(* Schneider Machine Expert - Basic project taffic_control_project, file version 1.8.0.0 *)
(* ProjectInformations: Name=New project *)

HARDWARE
  Cpu 0: TM221CE16R
  EthernetConfiguration: NetworkName=M221, IpAllocationMode=FixedAddress, IpAddress=0.0.0.0, SubnetMask=0.0.0.0
  SerialLineConfiguration: Baud=Baud19200, Parity=ParityEven, DataBits=DataBits8, StopBits=StopBits1, PhysicalMedium=PhysicalMediumRs485, TransmissionMode=TransmissionModeModbusRtu, SlaveId=1, Addressing=SlaveAddressing
  MastTask: UsePeriodScanMode=false, PeriodScan=100
  FastTask: Period=255
  CpuBehavior: StartingMode=StartAsPreviousState, AutoSaveRamOnEeprom=true, WatchdogPeriod=250

SYMBOLS  (address, symbol, comment, settings)
  %TM0        [Preset=1, Base=OneSecond, IsRetentive=true]
  %TM1        [Preset=1, Base=OneSecond, IsRetentive=true]
  %TM2        [Preset=5, Base=OneSecond, IsRetentive=true]
  %TM3        [Preset=3, Base=OneSecond, IsRetentive=true]
  %TM4        [Preset=3, Base=OneSecond, IsRetentive=true]
  %TM5        [Preset=3, Base=OneSecond, IsRetentive=true]
  %TM6        [Preset=3, Base=OneSecond, IsRetentive=true]

POU state
  (* SectionNumber=1 *)

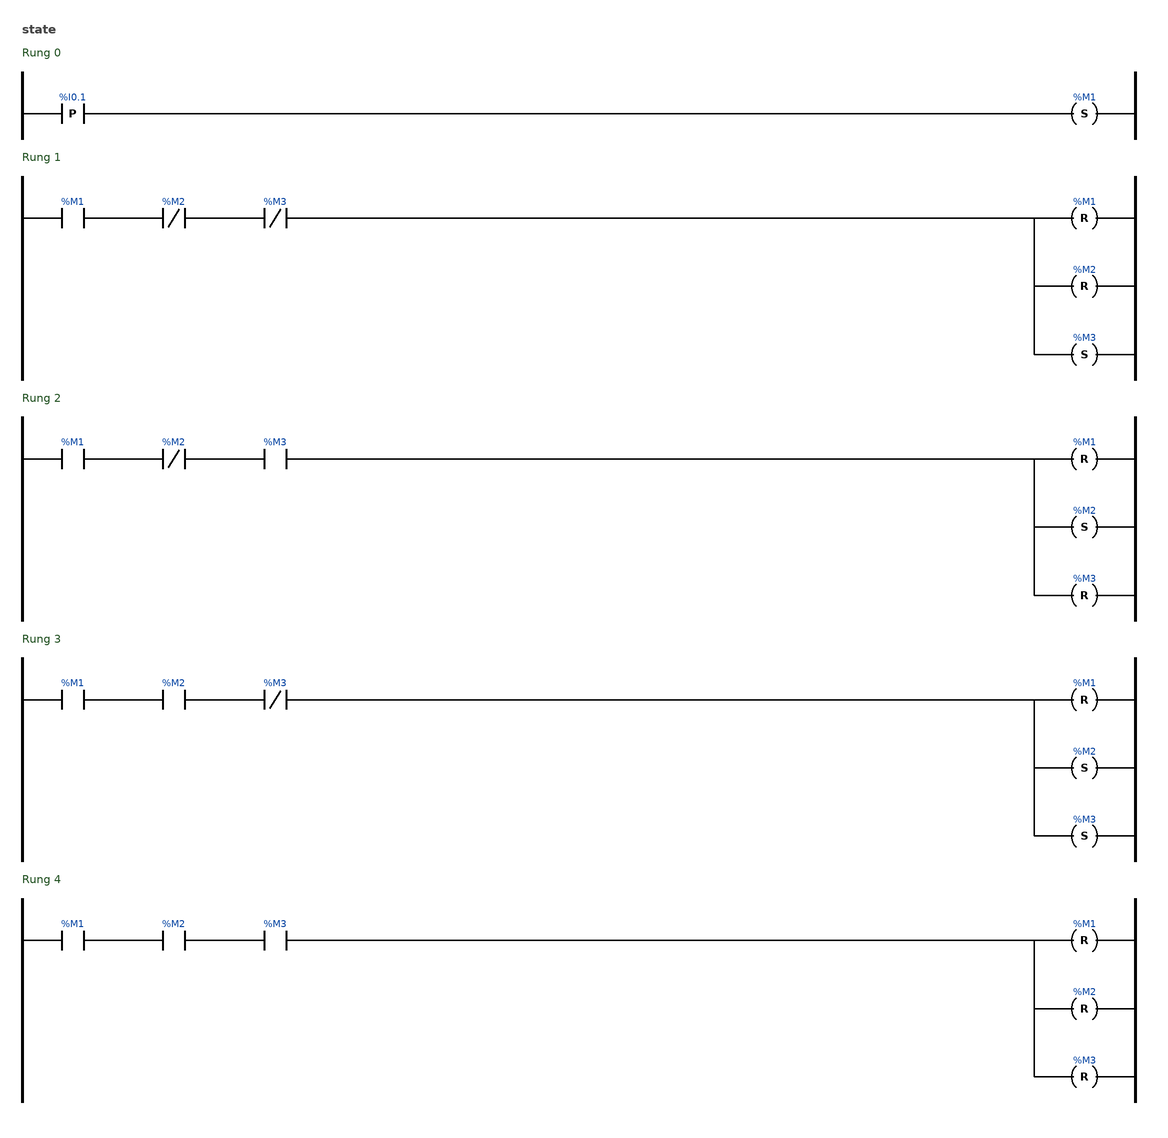

// Rung 0
  LDR %I0.1
  S %M1
  // as ST:
  //   IF RISING(%I0.1) THEN %M1 := TRUE; END_IF;

// Rung 1
  LD %M1
  ANDN %M2
  ANDN %M3
  R %M1
  R %M2
  S %M3
  // as ST:
  //   _t1 := %M1 AND NOT %M2 AND NOT %M3;
  //   IF _t1 THEN %M1 := FALSE; END_IF;
  //   IF _t1 THEN %M2 := FALSE; END_IF;
  //   IF _t1 THEN %M3 := TRUE; END_IF;

// Rung 2
  LD %M1
  ANDN %M2
  AND %M3
  R %M1
  S %M2
  R %M3
  // as ST:
  //   _t1 := %M1 AND NOT %M2 AND %M3;
  //   IF _t1 THEN %M1 := FALSE; END_IF;
  //   IF _t1 THEN %M2 := TRUE; END_IF;
  //   IF _t1 THEN %M3 := FALSE; END_IF;

// Rung 3
  LD %M1
  AND %M2
  ANDN %M3
  R %M1
  S %M2
  S %M3
  // as ST:
  //   _t1 := %M1 AND %M2 AND NOT %M3;
  //   IF _t1 THEN %M1 := FALSE; END_IF;
  //   IF _t1 THEN %M2 := TRUE; END_IF;
  //   IF _t1 THEN %M3 := TRUE; END_IF;

// Rung 4
  LD %M1
  AND %M2
  AND %M3
  R %M1
  R %M2
  R %M3
  // as ST:
  //   _t1 := %M1 AND %M2 AND %M3;
  //   IF _t1 THEN %M1 := FALSE; END_IF;
  //   IF _t1 THEN %M2 := FALSE; END_IF;
  //   IF _t1 THEN %M3 := FALSE; END_IF;

POU yello blink
  (* SectionNumber=2 *)

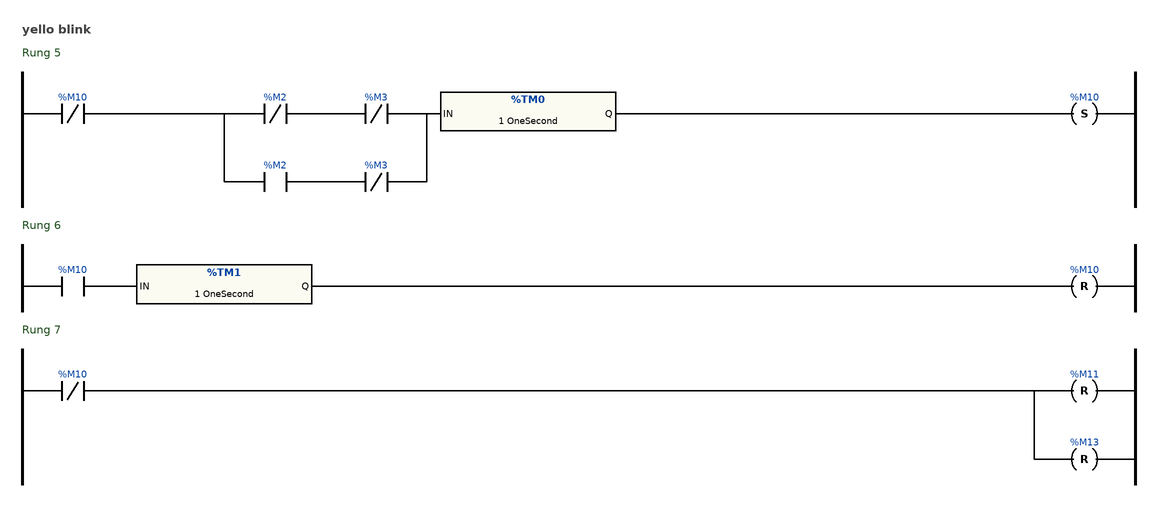

// Rung 5
  BLK %TM0
  LDN %M10
  AND(N %M2
  ANDN %M3
  OR( %M2
  ANDN %M3
  )
  )
  IN
  OUT_BLK
  LD Q
  S %M10
  END_BLK
  // as ST:
  //   %TM0(IN := NOT %M10 AND (NOT %M2 AND NOT %M3 OR %M2 AND NOT %M3));
  //   IF %TM0.Q THEN %M10 := TRUE; END_IF;

// Rung 6
  BLK %TM1
  LD %M10
  IN
  OUT_BLK
  LD Q
  R %M10
  END_BLK
  // as ST:
  //   %TM1(IN := %M10);
  //   IF %TM1.Q THEN %M10 := FALSE; END_IF;

// Rung 7
  LDN %M10
  R %M11
  R %M13
  // as ST:
  //   IF NOT %M10 THEN %M11 := FALSE; END_IF;
  //   IF NOT %M10 THEN %M13 := FALSE; END_IF;

POU Manual
  (* SectionNumber=3 *)

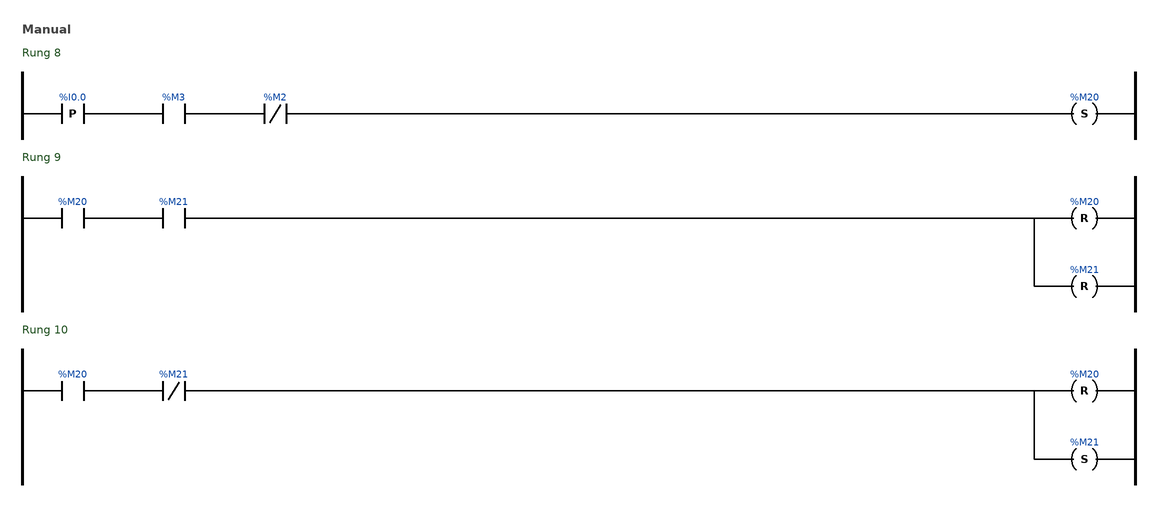

// Rung 8
  LDR %I0.0
  AND %M3
  ANDN %M2
  S %M20
  // as ST:
  //   IF RISING(%I0.0) AND %M3 AND NOT %M2 THEN %M20 := TRUE; END_IF;

// Rung 9
  LD %M20
  AND %M21
  R %M20
  R %M21
  // as ST:
  //   _t1 := %M20 AND %M21;
  //   IF _t1 THEN %M20 := FALSE; END_IF;
  //   IF _t1 THEN %M21 := FALSE; END_IF;

// Rung 10
  LD %M20
  ANDN %M21
  R %M20
  S %M21
  // as ST:
  //   _t1 := %M20 AND NOT %M21;
  //   IF _t1 THEN %M20 := FALSE; END_IF;
  //   IF _t1 THEN %M21 := TRUE; END_IF;

POU Manual_LED
  (* SectionNumber=4 *)

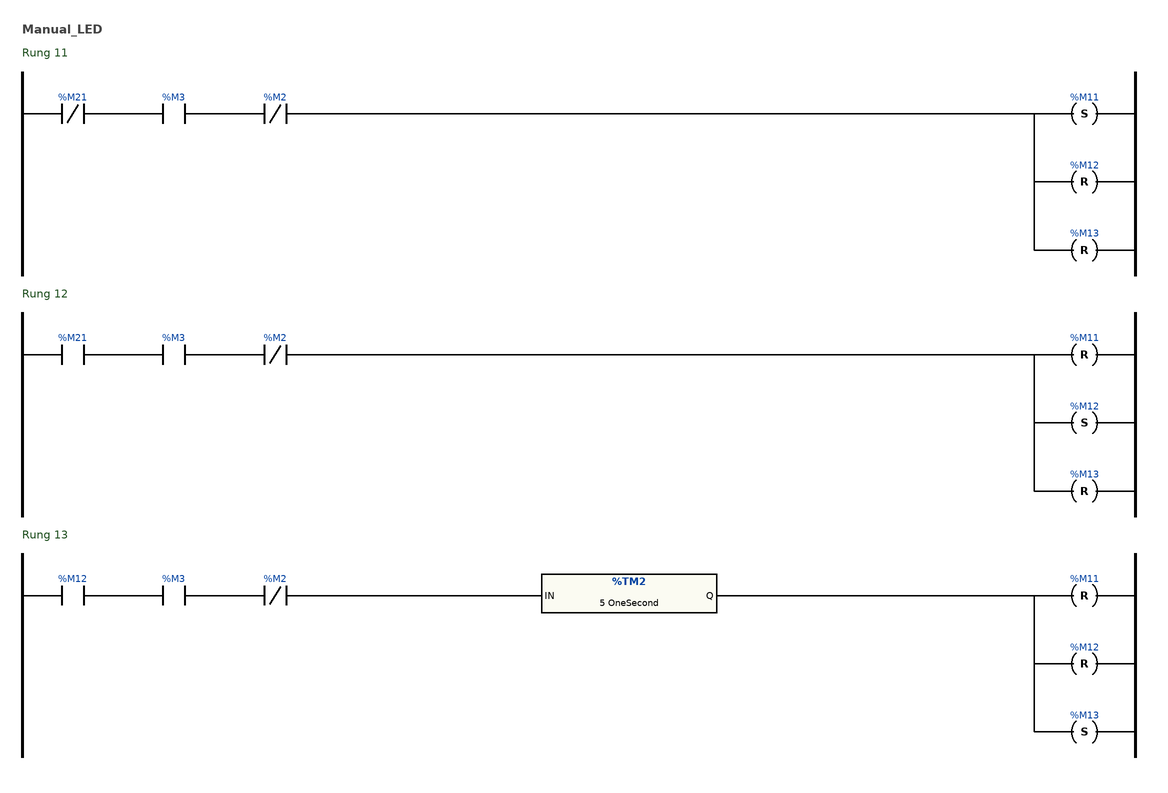

// Rung 11
  LDN %M21
  AND %M3
  ANDN %M2
  S %M11
  R %M12
  R %M13
  // as ST:
  //   IF NOT %M21 AND %M3 AND NOT %M2 THEN %M11 := TRUE; END_IF;
  //   IF NOT %M21 AND %M3 AND NOT %M2 THEN %M12 := FALSE; END_IF;
  //   IF NOT %M21 AND %M3 AND NOT %M2 THEN %M13 := FALSE; END_IF;

// Rung 12
  LD %M21
  AND %M3
  ANDN %M2
  R %M11
  S %M12
  R %M13
  // as ST:
  //   IF %M21 AND %M3 AND NOT %M2 THEN %M11 := FALSE; END_IF;
  //   IF %M21 AND %M3 AND NOT %M2 THEN %M12 := TRUE; END_IF;
  //   IF %M21 AND %M3 AND NOT %M2 THEN %M13 := FALSE; END_IF;

// Rung 13
  BLK %TM2
  LD %M12
  AND %M3
  ANDN %M2
  IN
  OUT_BLK
  LD Q
  R %M11
  R %M12
  S %M13
  END_BLK
  // as ST:
  //   %TM2(IN := %M12 AND %M3 AND NOT %M2);
  //   IF %TM2.Q THEN %M11 := FALSE; END_IF;
  //   IF %TM2.Q THEN %M12 := FALSE; END_IF;
  //   IF %TM2.Q THEN %M13 := TRUE; END_IF;

POU LED_Control
  (* SectionNumber=5 *)

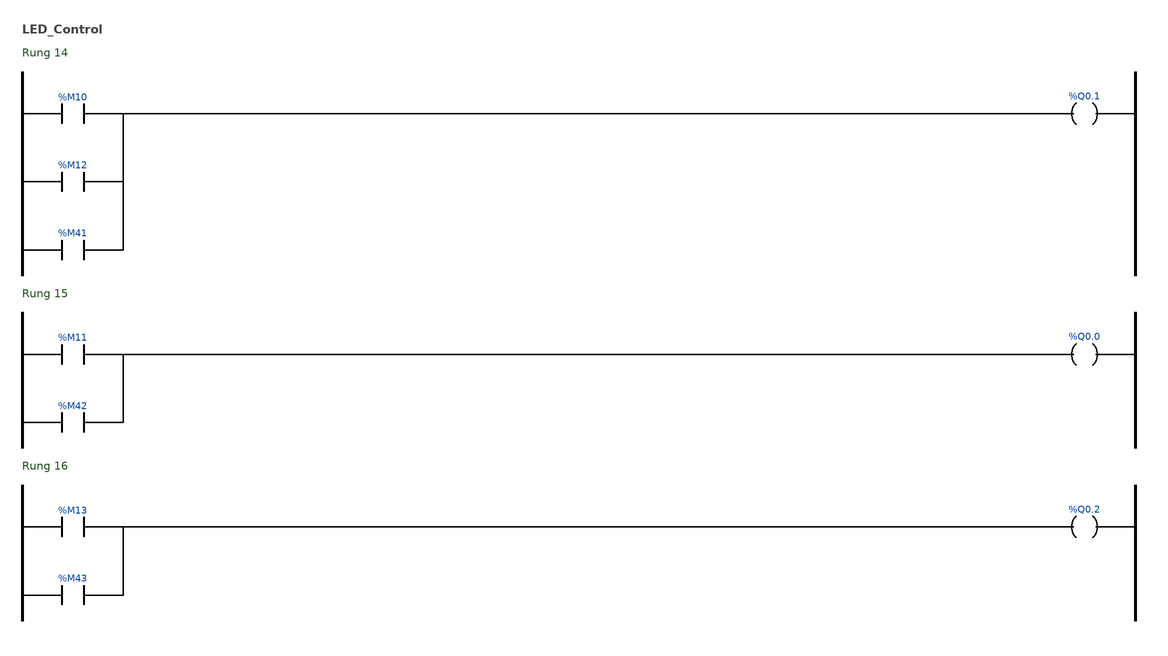

// Rung 14
  LD %M10
  OR %M12
  OR %M41
  ST %Q0.1
  // as ST:
  //   %Q0.1 := %M10 OR %M12 OR %M41;

// Rung 15
  LD %M11
  OR %M42
  ST %Q0.0
  // as ST:
  //   %Q0.0 := %M11 OR %M42;

// Rung 16
  LD %M13
  OR %M43
  ST %Q0.2
  // as ST:
  //   %Q0.2 := %M13 OR %M43;

POU Auto_Control
  (* SectionNumber=6 *)

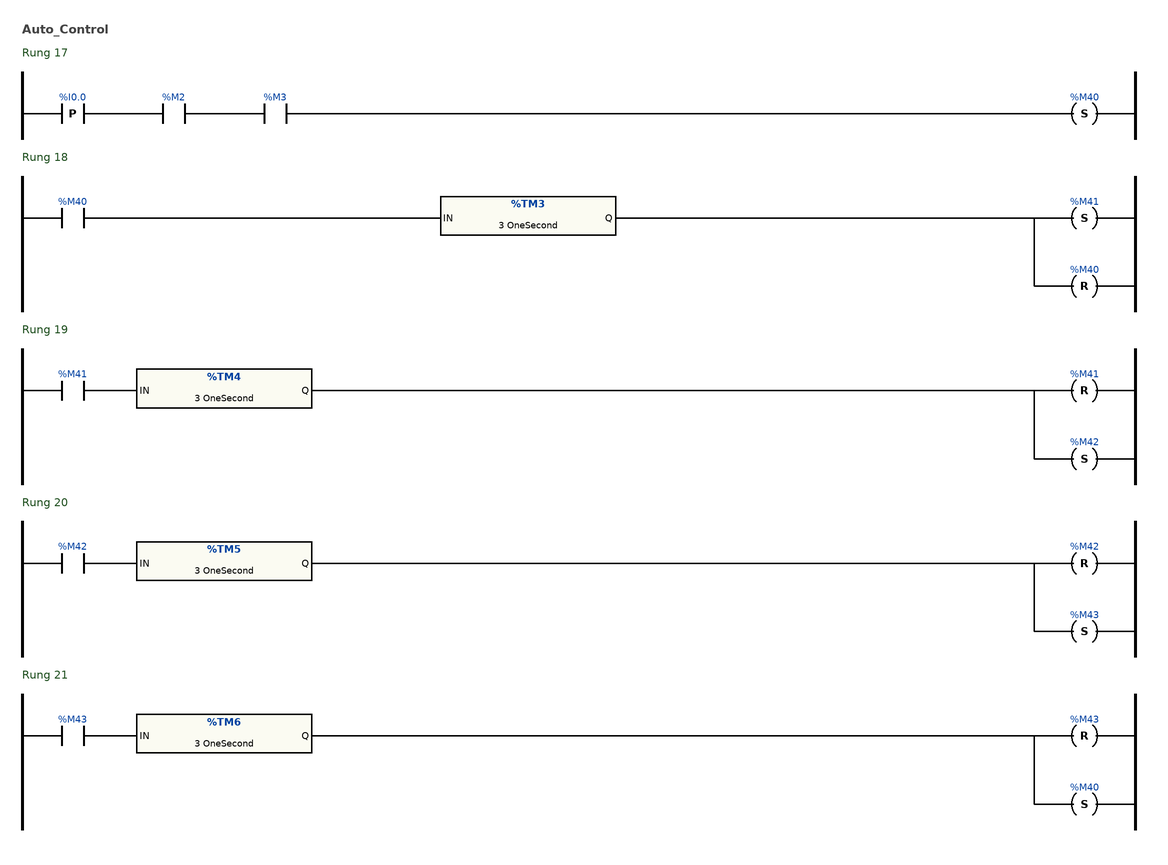

// Rung 17
  LDR %I0.0
  AND %M2
  AND %M3
  S %M40
  // as ST:
  //   IF RISING(%I0.0) AND %M2 AND %M3 THEN %M40 := TRUE; END_IF;

// Rung 18
  BLK %TM3
  LD %M40
  IN
  OUT_BLK
  LD Q
  S %M41
  R %M40
  END_BLK
  // as ST:
  //   %TM3(IN := %M40);
  //   IF %TM3.Q THEN %M41 := TRUE; END_IF;
  //   IF %TM3.Q THEN %M40 := FALSE; END_IF;

// Rung 19
  BLK %TM4
  LD %M41
  IN
  OUT_BLK
  LD Q
  R %M41
  S %M42
  END_BLK
  // as ST:
  //   %TM4(IN := %M41);
  //   IF %TM4.Q THEN %M41 := FALSE; END_IF;
  //   IF %TM4.Q THEN %M42 := TRUE; END_IF;

// Rung 20
  BLK %TM5
  LD %M42
  IN
  OUT_BLK
  LD Q
  R %M42
  S %M43
  END_BLK
  // as ST:
  //   %TM5(IN := %M42);
  //   IF %TM5.Q THEN %M42 := FALSE; END_IF;
  //   IF %TM5.Q THEN %M43 := TRUE; END_IF;

// Rung 21
  BLK %TM6
  LD %M43
  IN
  OUT_BLK
  LD Q
  R %M43
  S %M40
  END_BLK
  // as ST:
  //   %TM6(IN := %M43);
  //   IF %TM6.Q THEN %M43 := FALSE; END_IF;
  //   IF %TM6.Q THEN %M40 := TRUE; END_IF;
